FUNCTION TryConvert_TIME_TO_LINT : BOOL
VAR_INPUT
	in : TIME;
	out : REFERENCE TO LINT;
END_VAR

out := TIME_TO_LINT(in);
TryConvert_TIME_TO_LINT := TRUE;

END_FUNCTION

(* stored: Version 1.1.0.1, ProductVersion 3.1.4024.12
   POU TryConvert_TIME_TO_LINT: Id {5e0bb891-b8d9-4859-a22d-4884ebd4fdb1}, SpecialFunc None *)
